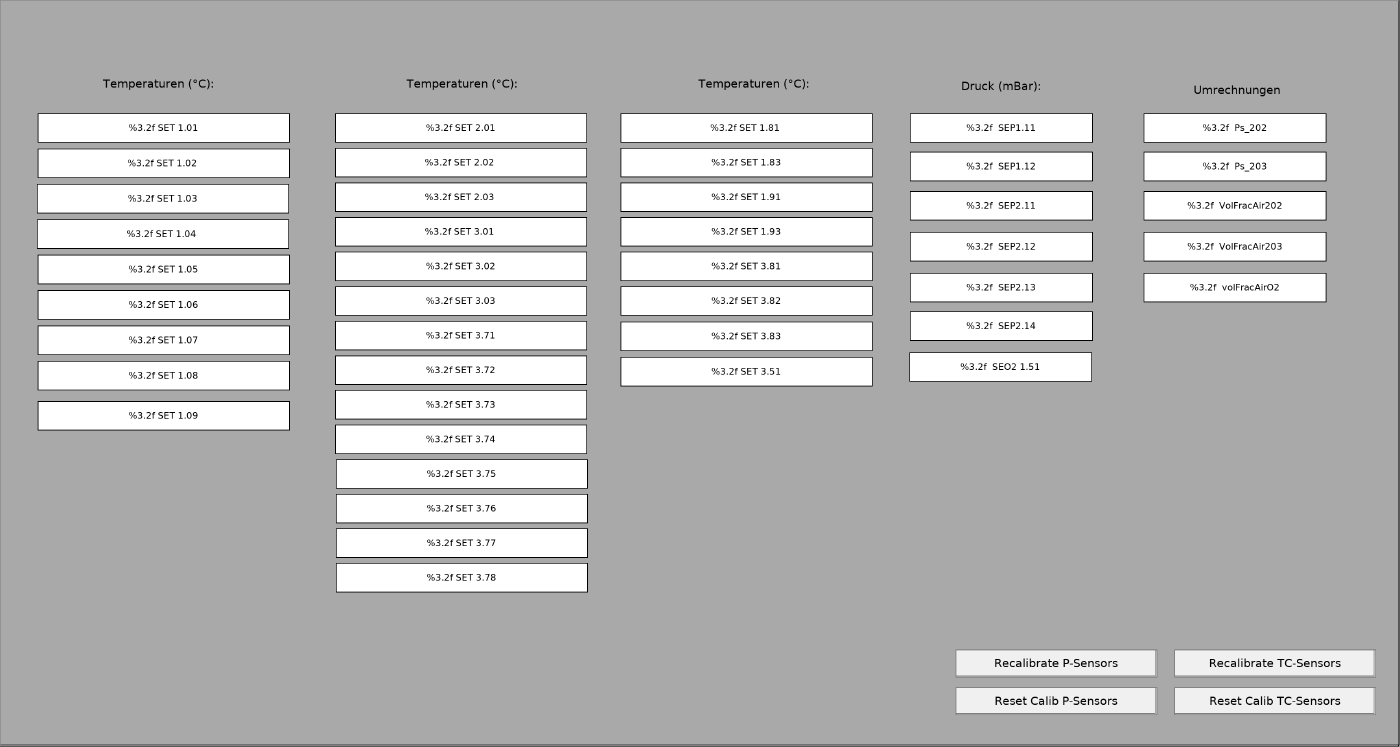
VISUALIZATION Sensors  // 1780x950
    Rectangle (48,144 320x37), "%3.2f SET 1.01", tooltip "Durchmesser in mm eingeben", text variable: GVL.T_Vor_WT_Visu
    Rectangle (48,189 320x37), "%3.2f SET 1.02", tooltip "Durchmesser in mm eingeben", text variable: GVL.T_nach_WT_Visu
    Rectangle (48,324 320x37), "%3.2f SET 1.05", tooltip "Durchmesser in mm eingeben", text variable: GVL.T_Einduesung_Oben_Visu
    Rectangle (48,369 320x37), "%3.2f SET 1.06", tooltip "Durchmesser in mm eingeben", text variable: GVL.T_Einduesung_Unten_Visu
    Rectangle (48,414 320x37), "%3.2f SET 1.07", tooltip "Durchmesser in mm eingeben", text variable: GVL.T_Absaugung_Oben_Visu
    Rectangle (48,459 320x37), "%3.2f SET 1.08", tooltip "Durchmesser in mm eingeben", text variable: GVL.T_Absaugung_Unten_Visu
    Rectangle (48,510 320x37), "%3.2f SET 1.09", tooltip "Durchmesser in mm eingeben", text variable: GVL.T_Vor_UmdampfLuefter_Visu
    Rectangle (120,94 164x25), "Temperaturen (°C):"
    Rectangle (1157,243 232x37), "%3.2f SEP2.11", tooltip "Durchmesser in mm eingeben", text variable: GVL.P_Komp_Einlass_Visu
    Rectangle (1203,97 140x25), "Druck (mBar):"
    Rectangle (1157,295 232x37), "%3.2f SEP2.12", tooltip "Durchmesser in mm eingeben", text variable: GVL.P_Komp_Auslass_Visu
    Rectangle (1157,144 232x37), "%3.2f SEP1.11", tooltip "Durchmesser in mm eingeben", text variable: GVL.P_Vor_WT_Visu
    Rectangle (1156,448 232x37), "%3.2f SEO2 1.51", tooltip "Durchmesser in mm eingeben", text variable: GVL.O2_Visu
    Rectangle (426,144 320x37), "%3.2f SET 2.01", tooltip "Durchmesser in mm eingeben", text variable: GVL.T_Komp_Einlass_Visu
    Rectangle (426,188 320x37), "%3.2f SET 2.02", tooltip "Durchmesser in mm eingeben", text variable: GVL.T_Komp_Auslass_Visu
    Rectangle (426,232 320x37), "%3.2f SET 2.03", tooltip "Durchmesser in mm eingeben", text variable: GVL.T_Kond_Auslass_Visu
    Rectangle (426,276 320x37), "%3.2f SET 3.01", tooltip "Durchmesser in mm eingeben", text variable: GVL.T_DK_Oben_Visu
    Rectangle (426,320 320x37), "%3.2f SET 3.02", tooltip "Durchmesser in mm eingeben", text variable: GVL.T_DK_Mitte_Visu
    Rectangle (426,364 320x37), "%3.2f SET 3.03", tooltip "Durchmesser in mm eingeben", text variable: GVL.T_DK_Unten_Visu
    Rectangle (426,408 320x37), "%3.2f SET 3.71", tooltip "Durchmesser in mm eingeben", text variable: GVL.T_Mat_Auslass1_Visu
    Rectangle (426,452 320x37), "%3.2f SET 3.72", tooltip "Durchmesser in mm eingeben", text variable: GVL.T_Mat_Auslass2_Visu
    Rectangle (426,496 320x37), "%3.2f SET 3.73", tooltip "Durchmesser in mm eingeben", text variable: GVL.T_Mat_Auslass3_Visu
    Rectangle (504,94 168x25), "Temperaturen (°C):"
    Rectangle (426,540 320x37), "%3.2f SET 3.74", tooltip "Durchmesser in mm eingeben", text variable: GVL.T_Mat_Auslass4_Visu
    Rectangle (789,144 320x37), "%3.2f SET 1.81", tooltip "Durchmesser in mm eingeben", text variable: GVL.T_DK_Band_oben1_Visu
    Rectangle (789,188 320x37), "%3.2f SET 1.83", tooltip "Durchmesser in mm eingeben", text variable: GVL.T_DK_Band_oben3_Visu
    Rectangle (789,232 320x37), "%3.2f SET 1.91", tooltip "Durchmesser in mm eingeben", text variable: GVL.T_DK_Band_unten1_Visu
    Rectangle (789,276 320x37), "%3.2f SET 1.93", tooltip "Durchmesser in mm eingeben", text variable: GVL.T_DK_Band_unten3_Visu
    Rectangle (789,320 320x37), "%3.2f SET 3.81", tooltip "Durchmesser in mm eingeben", text variable: GVL.T_DK_Steigband1_Visu
    Rectangle (874,94 170x25), "Temperaturen (°C):"
    Rectangle (789,364 320x37), "%3.2f SET 3.82", tooltip "Durchmesser in mm eingeben", text variable: GVL.T_DK_Steigband2_Visu
    Rectangle (789,409 320x37), "%3.2f SET 3.83", tooltip "Durchmesser in mm eingeben", text variable: GVL.T_DK_Steigband3_Visu
    Rectangle (1778,0 2x947)
    Rectangle (0,947 1778x3)
    Rectangle (427,584 320x37), "%3.2f SET 3.75", tooltip "Durchmesser in mm eingeben", text variable: GVL.T_Mat_Auslass5_Visu
    Rectangle (427,628 320x37), "%3.2f SET 3.76", tooltip "Durchmesser in mm eingeben", text variable: GVL.T_Mat_Auslass6_Visu
    Rectangle (427,672 320x37), "%3.2f SET 3.77", tooltip "Durchmesser in mm eingeben", text variable: GVL.T_Mat_Auslass7_Visu
    Rectangle (427,716 320x37), "%3.2f SET 3.78", tooltip "Durchmesser in mm eingeben", text variable: GVL.T_Mat_Auslass8_Visu
    Rectangle (47,234 320x37), "%3.2f SET 1.03", tooltip "Durchmesser in mm eingeben", text variable: T_HE_Einduesung_Oben_Visu
    Rectangle (47,279 320x37), "%3.2f SET 1.04", tooltip "Durchmesser in mm eingeben", text variable: T_HE_Einduesung_Unten_Visu
    Rectangle (1157,193 232x37), "%3.2f SEP1.12", tooltip "Durchmesser in mm eingeben", text variable: P_nach_WT_Visu
    Rectangle (1157,347 232x37), "%3.2f SEP2.13", tooltip "Durchmesser in mm eingeben", text variable: GVL.P_Kond_Auslass_Visu
    Rectangle (789,454 320x37), "%3.2f SET 3.51", tooltip "Durchmesser in mm eingeben", text variable: GVL.T_Komp_Gehaeuse_Visu
    Rectangle (1157,396 232x37), "%3.2f SEP2.14", tooltip "Durchmesser in mm eingeben", text variable: P_Abs_Amb_Visu
    Button (1493,826 256x35), "Recalibrate TC-Sensors", pressed state: GVL.Compressor_Switch_ON_Manu
        tap Re_Calibrate_TC
    Button (1493,874 256x35), "Reset Calib TC-Sensors", pressed state: GVL.Compressor_Switch_ON_Manu
        tap Reset_Calib
    Button (1215,826 256x35), "Recalibrate P-Sensors", pressed state: GVL.Compressor_Switch_ON_Manu
        tap Set_Calib_preasure
    Button (1215,874 256x35), "Reset Calib P-Sensors", pressed state: GVL.Compressor_Switch_ON_Manu
        tap Reset_Calib_preasure
    Rectangle (1454,243 232x37), "%3.2f VolFracAir202", tooltip "Durchmesser in mm eingeben", text variable: volFracAir202
    Rectangle (1454,295 232x37), "%3.2f VolFracAir203", tooltip "Durchmesser in mm eingeben", text variable: volFracAir203
    Rectangle (1454,144 232x37), "%3.2f Ps_202", tooltip "Durchmesser in mm eingeben", text variable: Ps_202
    Rectangle (1454,193 232x37), "%3.2f Ps_203", tooltip "Durchmesser in mm eingeben", text variable: Ps_203
    Rectangle (1454,347 232x37), "%3.2f volFracAirO2", tooltip "Durchmesser in mm eingeben", text variable: volFracAirO2
    Rectangle (1503,102 140x25), "Umrechnungen"
END_VISUALIZATION

(* stored: Version 1.1.0.1, ProductVersion 3.1.4024.3
   Visu Sensors: Id {36641c98-7e2f-444d-8d91-d35bf600eb1c} *)
